PROGRAM MAIN
VAR
	fb_Test_Conversion : Fb_AnalogToReal_Conversion;
	ntest: LREAL;
	fb_testR2A: Fb_RealToAnalog_Conversion;
	stTestString : STRING :='Added this for 1.0.1';
END_VAR

P_Test();
P_Feeder();
P_SheetAlignTable();
P_VacummBeltTable();
P_EjectionGate();
P_StackerBeltTable();
P_AllStateChecker();
P_GeneralStateManager();
//PRG_TEST();

fb_Test_Conversion(iRawVal:= , iMinVal:=0 , iMaxVal:=180 , lActualVal=>ntest );
fb_testR2A(lActualVal:= , lMinVal:=50 , lMaxVal:=100 , iRawVal=> );

//OOP Test
MAIN_OOP();

END_PROGRAM

(* stored: Version 1.1.0.1, ProductVersion 3.1.4024.12
   POU MAIN: Id {8bcade6c-ec1f-4118-bf4e-b1ed3c6ae3d8}, SpecialFunc None *)
